Fanuc KAREL source: ka00215.KL

-- PROVISIONAL review KL for V940-1; original PC SHA256 c5d374d33b9fe1ea5963e63deee48fe29bbf434d068d7ee598e46a15bbc182ab
-- Incomplete behavior may be omitted. Consult companion uncertainty JSON. Do not deploy.
PROGRAM KA00215
%NOLOCKGROUP
BEGIN
  -- V9_COMPOSED_GLOBAL_TRANSFER_HINT repetitions=1; address IDs observed; pairing/direction/source/runtime held
  -- V9_TWO_GLOBAL_ADDRESS_COPY_HINT bounded five-record physical form; type/direction/source/runtime held
  -- V9_ZERO_TABLE_METADATA_HINT layout=0001; no indexed target words; source/name/runtime held
  -- UNRESOLVED_PC offsets 5-19; opcodes 22,22,1E
  -- UNRESOLVED_PC offsets 24-28; opcodes 7F
END KA00215
